// SIMATIC S7-200 project (STEP 7-Micro/WIN), CPU 224 UN REL 02.01

SYMBOL_TABLE USER1
到下阀时间            VD500
到上阀时间            VD504
温度               VD508
成功与否             VD512
环境温度             VD516
END_SYMBOL_TABLE

ORGANIZATION_BLOCK 主程序:OB1
TITLE=PROGRAM COMMENTS
BEGIN
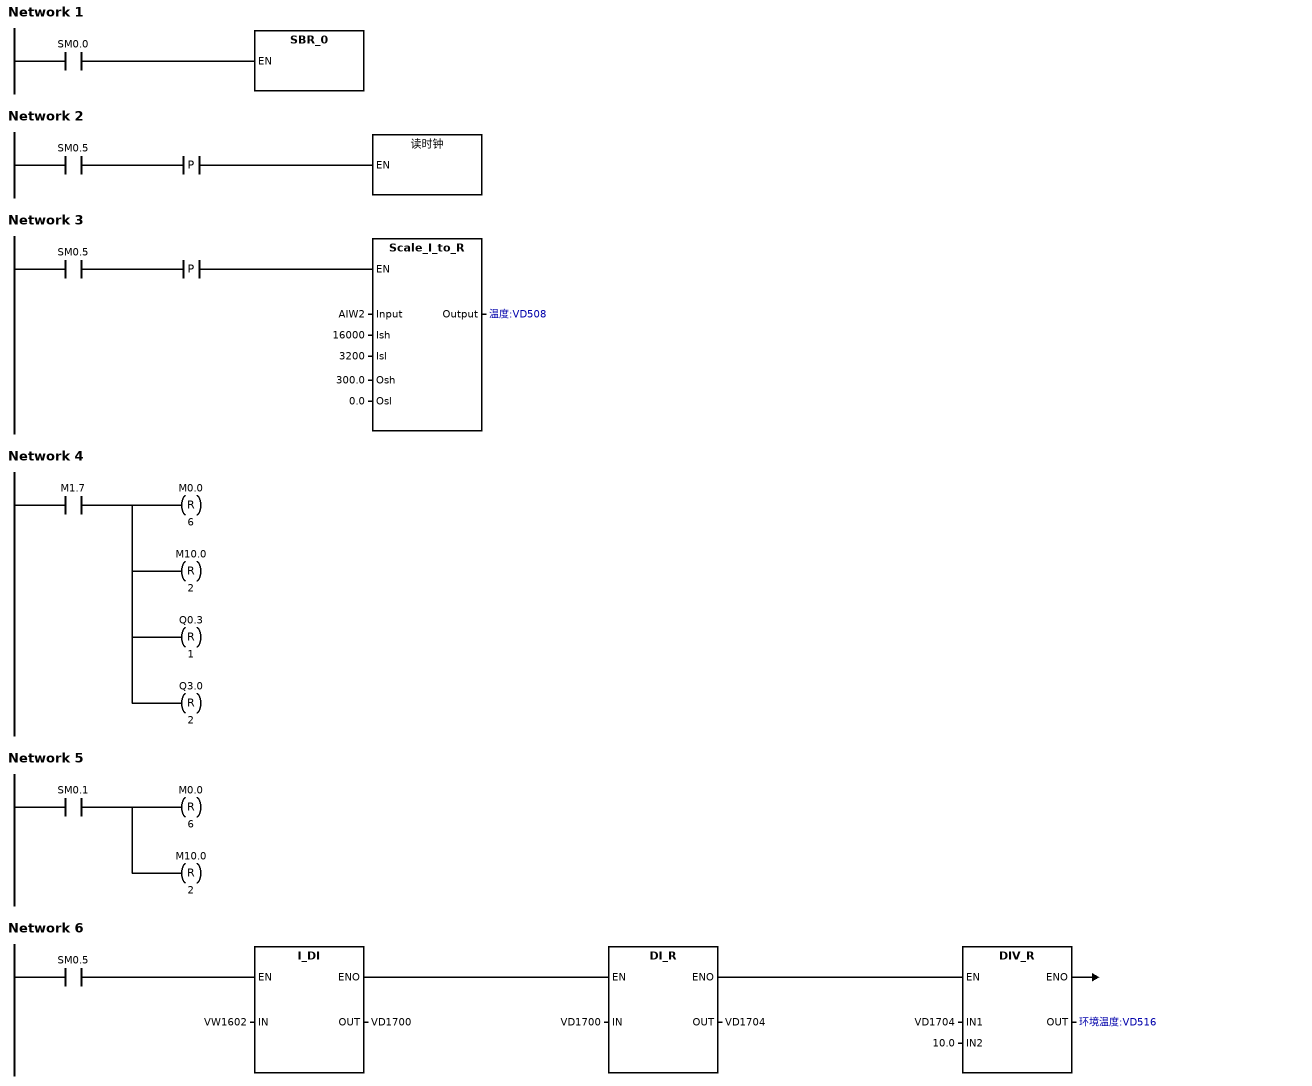
Network 1
LD     SM0.0
CALL   SBR_0:SBR0
Network 2
LD     SM0.5
EU
CALL   读时钟:SBR28
Network 3
LD     SM0.5
EU
CALL   Scale_I_to_R:SBR1, AIW2, 16000, 3200, 300.0, 0.0, 温度:VD508
Network 4
LD     M1.7
R      M0.0, 6
R      M10.0, 2
R      Q0.3, 1
R      Q3.0, 2
Network 5
LD     SM0.1
R      M0.0, 6
R      M10.0, 2
Network 6
LD     SM0.5
ITD    VW1602, VD1700
AENO
DTR    VD1700, VD1704
AENO
MOVR   VD1704, 环境温度:VD516
/R     10.0, 环境温度:VD516
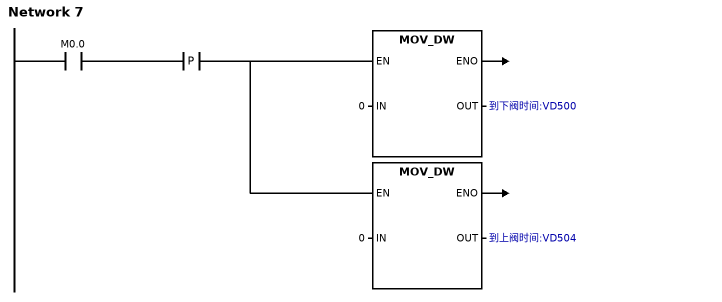
Network 7
LD     M0.0
EU
MOVD   0, 到下阀时间:VD500
MOVD   0, 到上阀时间:VD504
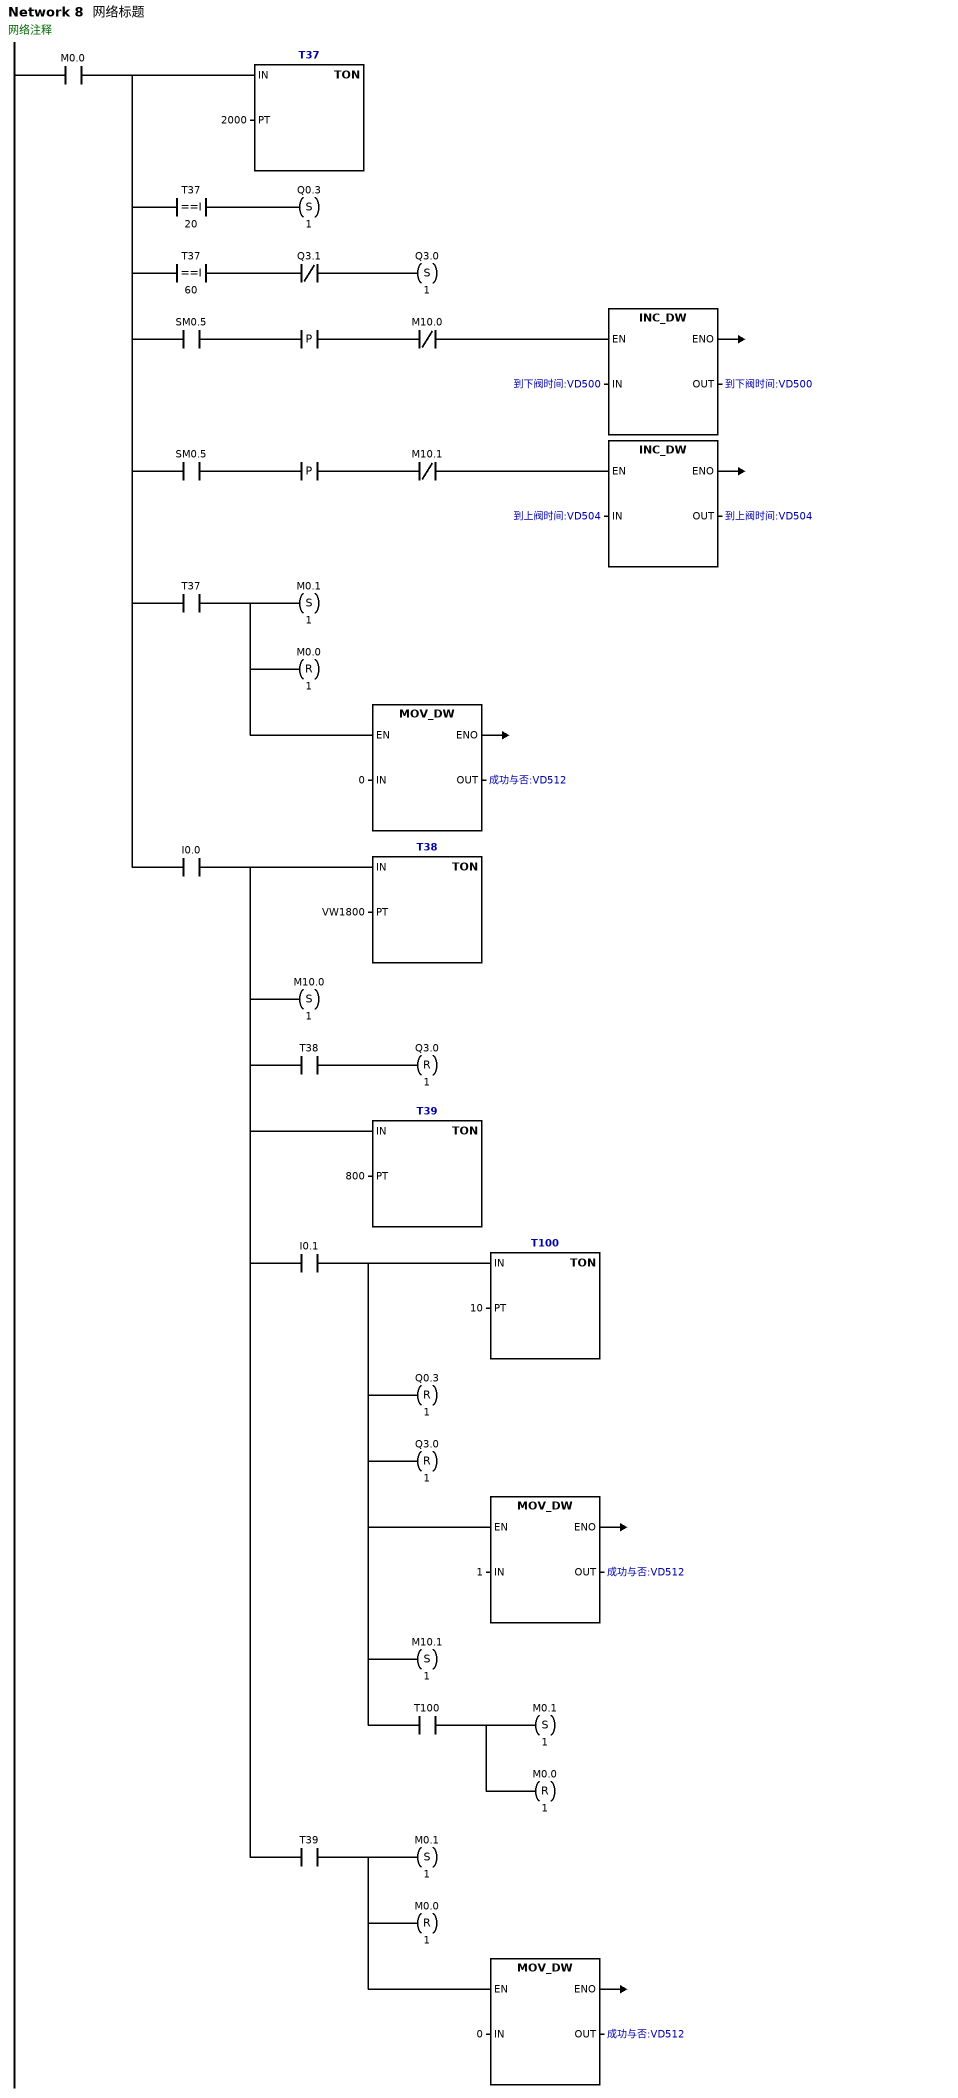
Network 8 // 网络标题
// 网络注释
LD     M0.0
LPS
TON    T37, 2000
AW=    T37, 20
S      Q0.3, 1
LRD
AW=    T37, 60
AN     Q3.1
S      Q3.0, 1
LRD
A      SM0.5
EU
AN     M10.0
INCD   到下阀时间:VD500
LRD
A      SM0.5
EU
AN     M10.1
INCD   到上阀时间:VD504
LRD
A      T37
S      M0.1, 1
R      M0.0, 1
MOVD   0, 成功与否:VD512
LPP
A      I0.0
LPS
TON    T38, VW1800
S      M10.0, 1
A      T38
R      Q3.0, 1
LRD
TON    T39, 800
LRD
A      I0.1
TON    T100, 10
R      Q0.3, 1
R      Q3.0, 1
MOVD   1, 成功与否:VD512
S      M10.1, 1
A      T100
S      M0.1, 1
R      M0.0, 1
LPP
A      T39
S      M0.1, 1
R      M0.0, 1
MOVD   0, 成功与否:VD512
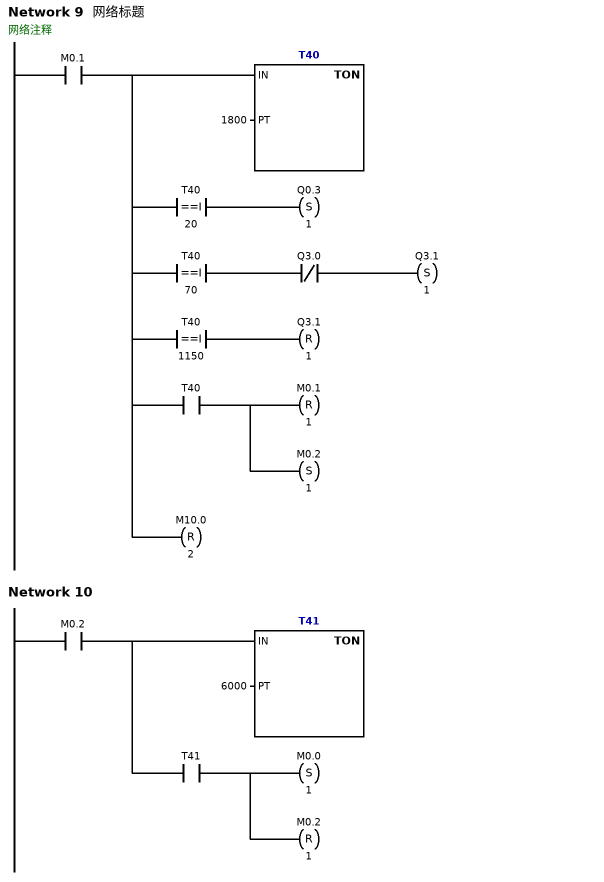
Network 9 // 网络标题
// 网络注释
LD     M0.1
LPS
TON    T40, 1800
AW=    T40, 20
S      Q0.3, 1
LRD
AW=    T40, 70
AN     Q3.0
S      Q3.1, 1
LRD
AW=    T40, 1150
R      Q3.1, 1
LRD
A      T40
R      M0.1, 1
S      M0.2, 1
LPP
R      M10.0, 2
Network 10
LD     M0.2
TON    T41, 6000
A      T41
S      M0.0, 1
R      M0.2, 1
END_ORGANIZATION_BLOCK

SUBROUTINE_BLOCK SBR_0:SBR0
TITLE=SUBROUTINE COMMENTS
BEGIN
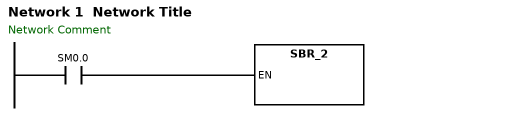
Network 1 // Network Title
// Network Comment
LD     SM0.0
CALL   SBR_2:SBR2
END_SUBROUTINE_BLOCK

// SBR1: protected block, not included

SUBROUTINE_BLOCK SBR_2:SBR2
TITLE=子程序注释
BEGIN
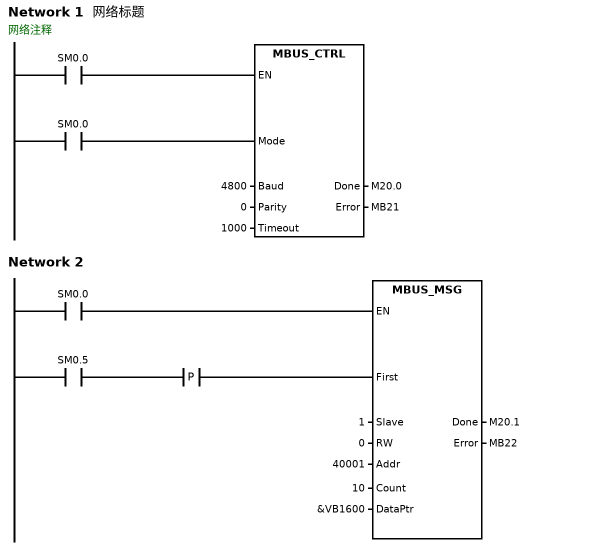
Network 1 // 网络标题
// 网络注释
LD     SM0.0
=      L60.0
LD     SM0.0
=      L63.7
LD     L60.0
CALL   MBUS_CTRL:SBR3, L63.7, 4800, 0, 1000, M20.0, MB21
Network 2
LD     SM0.0
=      L60.0
LD     SM0.5
EU
=      L63.7
LD     L60.0
CALL   MBUS_MSG:SBR4, L63.7, 1, 0, 40001, 10, &VB1600, M20.1, MB22
END_SUBROUTINE_BLOCK

// SBR3: protected block, not included

// SBR4: protected block, not included

SUBROUTINE_BLOCK 读时钟:SBR28
TITLE=
BEGIN
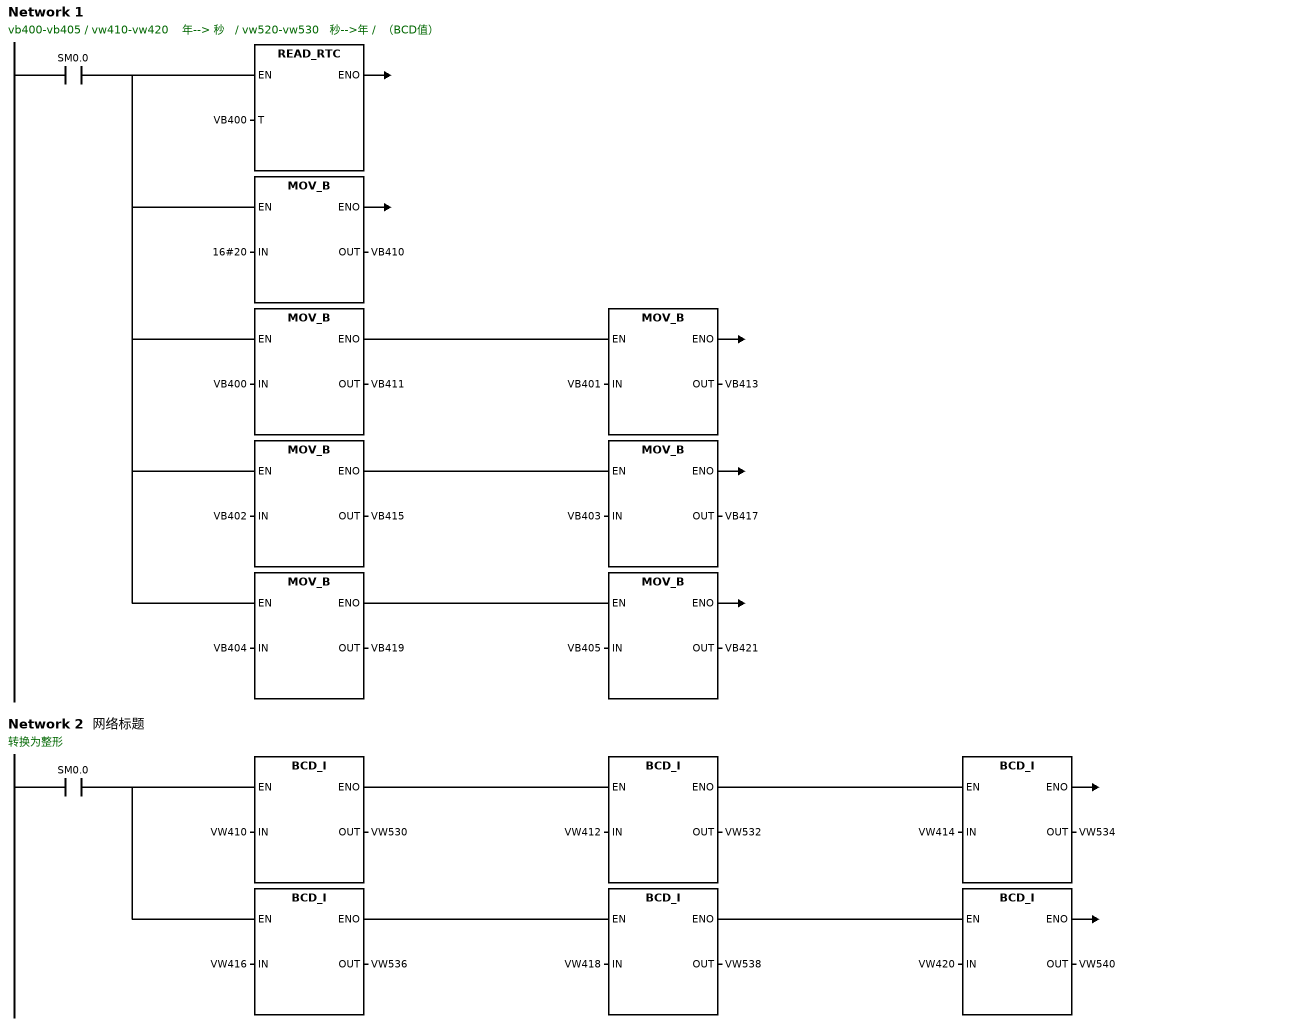
Network 1
// vb400-vb405
// vw410-vw420    年--> 秒  
// vw520-vw530   秒-->年
//  （BCD值）
LD     SM0.0
LPS
TODR   VB400
MOVB   16#20, VB410
MOVB   VB400, VB411
AENO
MOVB   VB401, VB413
LRD
MOVB   VB402, VB415
AENO
MOVB   VB403, VB417
LPP
MOVB   VB404, VB419
AENO
MOVB   VB405, VB421
Network 2 // 网络标题
// 转换为整形
LD     SM0.0
LPS
MOVW   VW410, VW530
AENO
BCDI   VW530
AENO
MOVW   VW412, VW532
AENO
BCDI   VW532
AENO
MOVW   VW414, VW534
BCDI   VW534
LPP
MOVW   VW416, VW536
AENO
BCDI   VW536
AENO
MOVW   VW418, VW538
AENO
BCDI   VW538
AENO
MOVW   VW420, VW540
BCDI   VW540
END_SUBROUTINE_BLOCK
